{attribute 'OPC.UA.DA.StructuredType' := '1'}
TYPE ST_ModuleAlarm :
STRUCT
	active			: BOOL;
	description		: STRING;
	level 			: E_FaultLevel;	
END_STRUCT
END_TYPE

(* stored: Version 1.1.0.1, ProductVersion 3.1.4024.13
   DUT ST_ModuleAlarm: Id {ca2c2b3d-6868-4bca-9876-84400760747c} *)
